INTERFACE I_TankController

METHOD ApplyCooling : BOOL
VAR_INPUT
END_VAR
END_METHOD

METHOD CheckSafety : BOOL
VAR_INPUT
END_VAR
END_METHOD

METHOD TransferChemical : BOOL
VAR_INPUT
END_VAR
END_METHOD

END_INTERFACE

(* stored: Version 1.1.0.1, ProductVersion 3.1.4024.16
   Itf I_TankController: Id {52460abf-02f3-42d1-9c4c-d4c5a8d3f5a8}
   Method ApplyCooling: Id {01367c06-4dea-4c49-9fe0-0829e57a8e88}
   Method CheckSafety: Id {577f5fb1-f3b7-49f8-b5f5-8ed3c73ae18d}
   Method TransferChemical: Id {a45b45a3-4497-4a7b-8b82-0e9f6c8c45c5} *)
